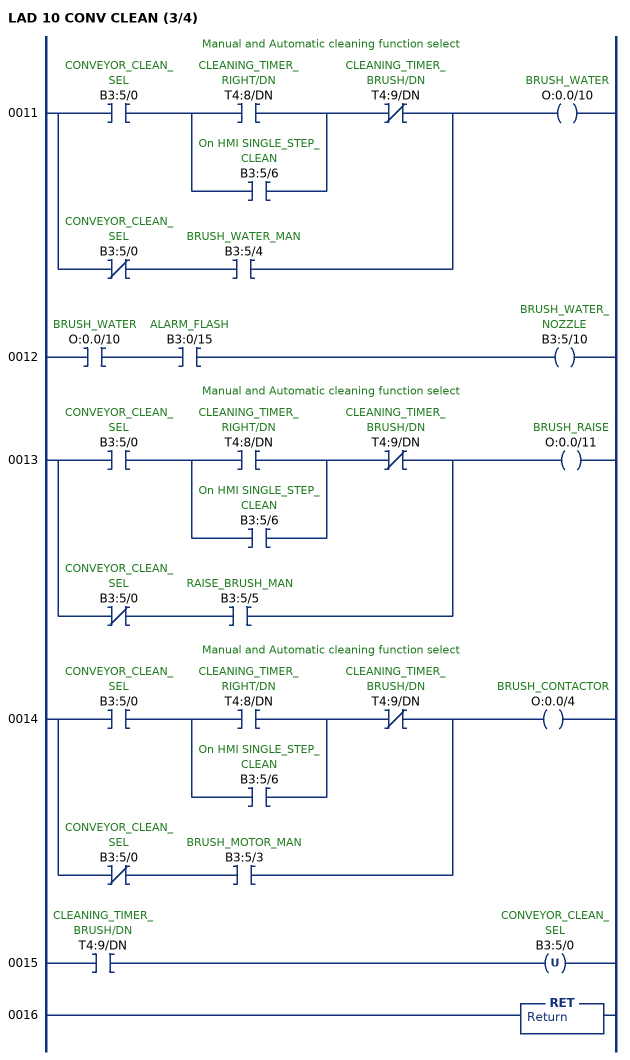
% Rung: 11 %
% Manual and Automatic cleaning function select %
SOR BST XIC B3:5/0 BST XIC T4:8/DN NXB XIC B3:5/6 BND XIO T4:9/DN NXB XIO B3:5/0 XIC B3:5/4 BND OTE O:0.0/10 EOR
%   B3:5/0  CONVEYOR_CLEAN_SEL %
%   T4:8  CLEANING_TIMER_RIGHT %
%   B3:5/6  SINGLE_STEP_CLEAN  "On HMI" %
%   T4:9  CLEANING_TIMER_BRUSH %
%   B3:5/4  BRUSH_WATER_MAN %
%   O:0.0/10  BRUSH_WATER %
% Rung: 12 %
SOR XIC O:0.0/10 XIC B3:0/15 OTE B3:5/10 EOR
%   O:0.0/10  BRUSH_WATER %
%   B3:0/15  ALARM_FLASH %
%   B3:5/10  BRUSH_WATER_NOZZLE %
% Rung: 13 %
% Manual and Automatic cleaning function select %
SOR BST XIC B3:5/0 BST XIC T4:8/DN NXB XIC B3:5/6 BND XIO T4:9/DN NXB XIO B3:5/0 XIC B3:5/5 BND OTE O:0.0/11 EOR
%   B3:5/0  CONVEYOR_CLEAN_SEL %
%   T4:8  CLEANING_TIMER_RIGHT %
%   B3:5/6  SINGLE_STEP_CLEAN  "On HMI" %
%   T4:9  CLEANING_TIMER_BRUSH %
%   B3:5/5  RAISE_BRUSH_MAN %
%   O:0.0/11  BRUSH_RAISE %
% Rung: 14 %
% Manual and Automatic cleaning function select %
SOR BST XIC B3:5/0 BST XIC T4:8/DN NXB XIC B3:5/6 BND XIO T4:9/DN NXB XIO B3:5/0 XIC B3:5/3 BND OTE O:0.0/4 EOR
%   B3:5/0  CONVEYOR_CLEAN_SEL %
%   T4:8  CLEANING_TIMER_RIGHT %
%   B3:5/6  SINGLE_STEP_CLEAN  "On HMI" %
%   T4:9  CLEANING_TIMER_BRUSH %
%   B3:5/3  BRUSH_MOTOR_MAN %
%   O:0.0/4  BRUSH_CONTACTOR %
% Rung: 15 %
SOR XIC T4:9/DN OTU B3:5/0 EOR
%   T4:9  CLEANING_TIMER_BRUSH %
%   B3:5/0  CONVEYOR_CLEAN_SEL %
% Rung: 16 %
SOR RET EOR

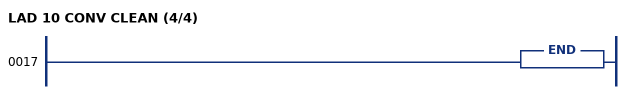
% Rung: 17 %
SOR END EOR

LADDER 11 "FAULTS"
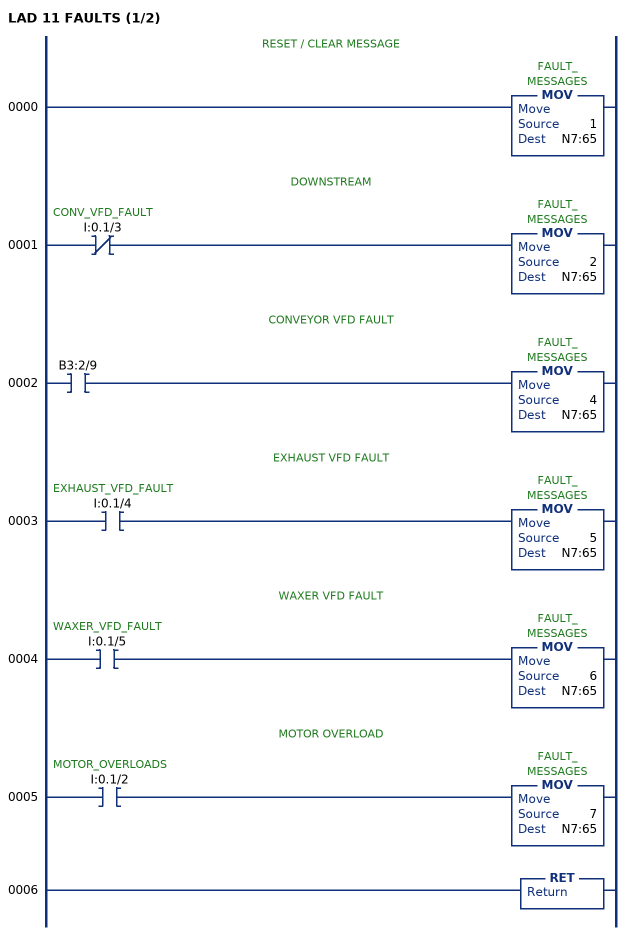
% Rung: 0 %
% RESET / CLEAR MESSAGE %
SOR MOV 1 N7:65 EOR
%   N7:65  FAULT_MESSAGES %
% Rung: 1 %
% DOWNSTREAM %
SOR XIO I:0.1/3 MOV 2 N7:65 EOR
%   I:0.1/3  CONV_VFD_FAULT %
%   N7:65  FAULT_MESSAGES %
% Rung: 2 %
% CONVEYOR VFD FAULT %
SOR XIC B3:2/9 MOV 4 N7:65 EOR
%   N7:65  FAULT_MESSAGES %
% Rung: 3 %
% EXHAUST VFD FAULT %
SOR XIC I:0.1/4 MOV 5 N7:65 EOR
%   I:0.1/4  EXHAUST_VFD_FAULT %
%   N7:65  FAULT_MESSAGES %
% Rung: 4 %
% WAXER VFD FAULT %
SOR XIC I:0.1/5 MOV 6 N7:65 EOR
%   I:0.1/5  WAXER_VFD_FAULT %
%   N7:65  FAULT_MESSAGES %
% Rung: 5 %
% MOTOR OVERLOAD %
SOR XIC I:0.1/2 MOV 7 N7:65 EOR
%   I:0.1/2  MOTOR_OVERLOADS %
%   N7:65  FAULT_MESSAGES %
% Rung: 6 %
SOR RET EOR

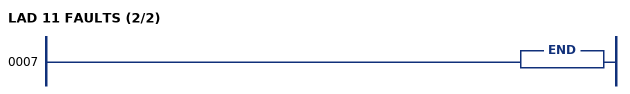
% Rung: 7 %
SOR END EOR

OTHER DOCUMENTED ADDRESSES
  B3:0/14  SET_MIN_VFD_SPEED
  B3:1/15  CONV_TEMP_INTERLOCK
  B3:4/5  DISPLAY_CNT_ON_TIME
  B3:5/15  POP_UP_SCREEN  "On HMI"
  I:0.0/12  VERI_FLAME_IGNITION
  I:0.0/14  VALVE_PROVING_ALARM
  I:0.0/15  REMOTE_START
  I:1.0/0  TC1
  I:2.0/0  SENSOR_PLENUM
  I:2.0/1  SENSOR_RETURN
  I:2.1/0  SENSOR_Q
  I:2.2/0  SENSOR_HUMIDITY
  I:2.3/0  SENSOR_TEMP_RHL
  N7:30  PV_RH_PROCESS_VAR  "Feedback from humidity sensors - calculated value"
  N7:38  SCALLED_RH_FOR_LOGGI
  N7:46  PLENUM_PS_ALARM
  N7:59  SCALLED_SPEED_REF
  N7:63  TEMP_SET_POINT  "For conveyor start"
  PD9:0.3  "SPS Setpoint"
  PFILE:5  "a"
  PFILE:10  "Brush Clening"
  T4:6  EXHAUST_INV_POWERUP

COMMENTS NOT ATTACHED TO A CURRENT RUNG
  N7:3: Subract to bring sensor value to zero
  N7:65: CONVEYOR VFD FAULT
  N7:50: Find slope step #2 -  multiply Y dif by 100 to get better accuracy
  N7:52: Multiply RH difference by Speed Scaller
  N7:53: Find slope intercept  b value step #2 -  multiply point Ax times slope
  N7:54: Find slope intercept  b value step #3 -  multiply point Ay by 100 for Accuracy
  N7:55: Find slope intercept  b value step #5 -  sub Ay minus Ax*slope
  N7:56: Solve for speed Step #2 - divide by 100 (multiply slope times humidity)
  N7:0: Read input card - Return Pressure
  N7:5: Read input card - Return Pressure
  O:3.1: With PID on, set max speed independent to PID

DATA TABLE (non-zero values as saved)
DATA B3
% B3:0 % 0X300D 0X43FF 0X01FF 0X0001 0X0480 0X0000
DATA T4
% .PRE .ACC %
% T4:0 % 3599 1744
% T4:1 % 1 0
% T4:2 % 150 139
% T4:3 % 100 0
% T4:4 % 3600 1788
% T4:5 % 10 0
% T4:6 % 4 0
% T4:7 % 60 0
% T4:8 % 60 0
% T4:9 % 60 0
% T4:10 % 9999 0
DATA N7
% N7:0 % 7402 6185 100 1 5 6312 6240 396 0 1
% N7:10 % 507 503 499 1509 200 1700 1500 1509 5272 8000
% N7:20 % 8990 6250 170 0 19 25 300 50 75 12
% N7:30 % 0 0 0 9776 13027 60 3599 151 4 0
% N7:40 % 4 8 4 100 0 5 0 0 0 0
% N7:50 % 0 0 0 0 55 1 20 20 0 0
% N7:60 % 10 0 0 90 0 1 691 0 0 0
% N7:70 % 1 1 1 0 0 0 0 0 0 0
DATA F8
% F8:0 % 45
